TYPE U_MOVER_SELECTOR_CTRL :
UNION
  stCtrl              : ST_MOVER_SELECTOR_CTRL;

  byCtrl    AT %I*    : ARRAY[1..SIZEOF(ST_MOVER_SELECTOR_CTRL)] OF BYTE;

END_UNION
END_TYPE

(* stored: Version 1.1.0.1, ProductVersion 3.1.4026.13
   DUT U_MOVER_SELECTOR_CTRL: Id {2f53cd33-953c-4a60-8a36-fa2601bc558c} *)
